// Mitsubishi GX Works2 project: BookEX6_48 Analog   PLC: Q13UDV

// global labels: Global
VAR_GLOBAL
  bVar0 AT M5000 : BOOL;
  abArray0 AT M5010 : ARRAY [0..49] OF BOOL;
  sStr0 AT D5000 : STRING[199];
  sStr1 AT D5100 : STRING[199];
  sStr2 AT D5200 : STRING[199];
  sStr3 AT D5300 : STRING[199];
  sStr4 AT D5400 : STRING[199];
  sStr5 AT D5500 : STRING[199];
  sStr6 AT D5600 : STRING[199];
  sStr7 AT D5700 : STRING[199];
  sStr8 AT D5800 : STRING[199];
  sStr9 AT D5900 : STRING[199];
  iVar0 AT D4500 : INT;
  iVar1 AT D4501 : INT;
  iVar2 AT D4502 : INT;
  iVar3 AT D4503 : INT;
  iVar4 AT D4504 : INT;
  iVar5 AT D4505 : INT;
  iVar6 AT D4506 : INT;
  iVar7 AT D4507 : INT;
  iVar8 AT D4508 : INT;
  iVar9 AT D4509 : INT;
  dVar0 AT D4510 : DINT;
  dVar1 AT D4512 : DINT;
  dVar2 AT D4514 : DINT;
  dVar3 AT D4516 : DINT;
  dVar4 AT D4518 : DINT;
  dVar5 AT D4520 : DINT;
  dVar6 AT D4522 : DINT;
  dVar7 AT D4524 : DINT;
  dVar8 AT D4526 : DINT;
  dVar9 AT D4528 : DINT;
  wVar0 AT D4530 : WORD;
  wVar1 AT D4531 : WORD;
  wVar2 AT D4532 : WORD;
  wVar3 AT D4533 : WORD;
  wVar4 AT D4534 : WORD;
  wVar5 AT D4535 : WORD;
  wVar6 AT D4536 : WORD;
  wVar7 AT D4537 : WORD;
  wVar8 AT D4538 : WORD;
  wVar9 AT D4539 : WORD;
  dwVar0 AT D4540 : DWORD;
  dwVar1 AT D4542 : DWORD;
  dwVar2 AT D4544 : DWORD;
  dwVar3 AT D4546 : DWORD;
  dwVar4 AT D4548 : DWORD;
  dwVar5 AT D4550 : DWORD;
  dwVar6 AT D4552 : DWORD;
  dwVar7 AT D4554 : DWORD;
  dwVar8 AT D4556 : DWORD;
  dwVar9 AT D4558 : DWORD;
  fsVar0 AT D4560 : REAL;
  fsVar1 AT D4562 : REAL;
  fsVar2 AT D4564 : REAL;
  fsVar3 AT D4566 : REAL;
  fsVar4 AT D4568 : REAL;
  fsVar5 AT D4570 : REAL;
  fsVar6 AT D4572 : REAL;
  fsVar7 AT D4574 : REAL;
  fsVar8 AT D4576 : REAL;
  fsVar9 AT D4578 : REAL;
  fdVar0 AT D4580 : LREAL;
  tTime0 AT D4620 : TIME;
  tTime1 AT D4622 : TIME;
  tTime2 AT D4624 : TIME;
  tTime3 AT D4626 : TIME;
  tTime4 AT D4628 : TIME;
  tTime5 AT D4630 : TIME;
  tTime6 AT D4632 : TIME;
  tTime7 AT D4634 : TIME;
  tTime8 AT D4636 : TIME;
  tTime9 AT D4638 : TIME;
  tTime10 AT D4640 : TIME;
  bVar1 AT M5001 : BOOL;
  bVar2 AT M5002 : BOOL;
  bVar3 AT M5003 : BOOL;
  bVar4 AT M5004 : BOOL;
  bVar5 AT M5005 : BOOL;
  bVar6 AT M5006 : BOOL;
  bVar7 AT M5007 : BOOL;
  bVar8 AT M5008 : BOOL;
  bVar9 AT M5009 : BOOL;
  abArray1 AT M5060 : ARRAY [0..49] OF BOOL;
  abArray2 AT M5110 : ARRAY [0..49] OF BOOL;
  abArray3 AT M5160 : ARRAY [0..49] OF BOOL;
  abArray4 AT M5210 : ARRAY [0..49] OF BOOL;
  abArray5 AT M5260 : ARRAY [0..49] OF BOOL;
  abArray6 AT M5310 : ARRAY [0..49] OF BOOL;
  abArray7 AT M5360 : ARRAY [0..49] OF BOOL;
  abArray8 AT M5410 : ARRAY [0..49] OF BOOL;
  abArray9 AT M5460 : ARRAY [0..49] OF BOOL;
  fdVar1 AT D4584 : LREAL;
  fdVar2 AT D4588 : LREAL;
  fdVar3 AT D4592 : LREAL;
  fdVar4 AT D4596 : LREAL;
  fdVar5 AT D4600 : LREAL;
  fdVar6 AT D4604 : LREAL;
  fdVar7 AT D4608 : LREAL;
  fdVar8 AT D4612 : LREAL;
  fdVar9 AT D4616 : LREAL;
  afsPen0 AT D2000 : ARRAY [0..499] OF REAL;
  afsPen1 AT D3000 : ARRAY [0..499] OF REAL;
END_VAR
// user libraries (not included): HMI

FUNCTION_BLOCK adcRead
VAR_INPUT
  i_StartIO : INT;
  i_NoCh : INT;
  b_Reset : BOOL;
END_VAR
VAR_IN_OUT
  b_InitDone : BOOL;
END_VAR
VAR_OUTPUT
  b_Ready : BOOL;
  b_Error : BOOL;
END_VAR
VAR
  Buffer : ARRAY [0..15] OF WORD;
  bRes : BOOL;
  ix : INT;
  SeqInit : INT;
END_VAR
VAR_INPUT
  b_EN : BOOL;
END_VAR
VAR_OUTPUT
  b_ENO : BOOL;
  aw_Setup : ARRAY [0..7] OF WORD;
  ai_Value : ARRAY [0..7] OF INT;
END_VAR
;
b_ENO := b_EN;
IF NOT b_EN THEN
	RETURN;
END_IF;

(* Status *)
Z0 := i_StartIO * 16;
b_Error := X0FZ0;
b_Ready := X00Z0;

(* Reset *)
IF Y0FZ0 AND NOT b_Error THEN Y0FZ0 := FALSE; END_IF;
IF LDP(TRUE, b_Reset) THEN
	SeqInit := 0;
	b_InitDone := FALSE;
	IF b_Error THEN Y0FZ0 := TRUE; END_IF;
END_IF;

CASE SeqInit OF
	0 : 
		IF NOT b_InitDone AND NOT b_Error AND 1 <= i_NoCh AND  i_NoCh <= 8 THEN
			SeqInit := 1;
		END_IF;
	1 : 
		IF b_Ready THEN
			(* Config Setting Read *)
			bRes := FROM(TRUE , i_StartIO , 20 , 2 , Buffer[0]);
			CASE i_NoCh OF
				2 : 
					aw_Setup[0] := Buffer[0] AND 16#000F;
					aw_Setup[1] := Buffer[0] AND 16#00F0;
				4 : 
					aw_Setup[0] := Buffer[0] AND 16#000F;
					aw_Setup[1] := Buffer[0] AND 16#00F0;
					aw_Setup[2] := Buffer[0] AND 16#0F00;
					aw_Setup[3] := Buffer[0] AND 16#F000;
				8 : 
					aw_Setup[0] := Buffer[0] AND 16#000F;
					aw_Setup[1] := Buffer[0] AND 16#00F0;
					aw_Setup[2] := Buffer[0] AND 16#0F00;
					aw_Setup[3] := Buffer[0] AND 16#F000;
					aw_Setup[4] := Buffer[1] AND 16#000F;
					aw_Setup[5] := Buffer[1] AND 16#00F0;
					aw_Setup[6] := Buffer[1] AND 16#0F00;
					aw_Setup[7] := Buffer[1] AND 16#F000;
			END_CASE;
			SeqInit := 2;
		END_IF;
	2 : 
		b_InitDone := TRUE;
		SeqInit := 100;
END_CASE;

IF b_InitDone AND b_Ready AND X0EZ0 THEN
	bRes := FROM(TRUE , i_StartIO , 11 , 8 , Buffer[0]);
	FOR ix := 0 TO i_NoCh-1 BY 1 DO
		IF (Buffer[ix] AND 16#8000) = 16#8000 THEN
			ai_Value[ix] := -WORD_TO_INT(Buffer[ix] AND 16#7FFF);
		ELSE
			ai_Value[ix] := WORD_TO_INT(Buffer[ix] AND 16#7FFF);
		END_IF;
	END_FOR;
END_IF;
END_FUNCTION_BLOCK

FUNCTION_BLOCK adcRead1Ch
VAR_INPUT
  i_Ch : INT;
END_VAR
VAR
  iStatus : INT;
  bRes : BOOL;
END_VAR
VAR_INPUT
  b_EN : BOOL;
END_VAR
VAR_OUTPUT
  b_ENO : BOOL;
END_VAR
VAR_INPUT
  i_StartIO : INT;
END_VAR
VAR_OUTPUT
  b_Error : BOOL;
  i_ErrNo : INT;
  b_OK : BOOL;
END_VAR
VAR
  bReady : BOOL;
END_VAR
VAR_OUTPUT
  i_Value : INT;
END_VAR
VAR
  bStatus : BOOL;
END_VAR
;
b_ENO := b_EN;
IF NOT b_EN THEN
	b_OK := FALSE;
	b_Error := FALSE;
	i_ErrNo := 0;
	RETURN;
END_IF;
IF i_Ch < 1 OR i_Ch > 8 THEN
	b_OK := FALSE;
	b_Error := TRUE;
	i_Value := 0;
	i_ErrNo := 10;
	RETURN;
END_IF;
	
Z0 := i_StartIO * 16;
b_Error := X0FZ0;
bReady := X00Z0;
FROM(TRUE , i_StartIO , 10 , 1 , iStatus);
TEST(TRUE, iStatus, i_Ch-1, bStatus);

IF bReady  AND bStatus THEN 
	FROM(TRUE , i_StartIO , 10+i_Ch, 1 , iStatus);
	i_Value := iStatus;
	b_OK := TRUE;
	i_ErrNo := 0;
END_IF;
END_FUNCTION_BLOCK

FUNCTION_BLOCK adcScaling
VAR_INPUT
  i_Ch : INT;
END_VAR
VAR
  wStatus : INT;
  bRes : BOOL;
END_VAR
VAR_INPUT
  b_EN : BOOL;
END_VAR
VAR_OUTPUT
  b_ENO : BOOL;
END_VAR
VAR_INPUT
  i_StartIO : INT;
END_VAR
VAR_OUTPUT
  b_Error : BOOL;
  i_ErrNo : INT;
  b_OK : BOOL;
END_VAR
VAR
  bReady : BOOL;
END_VAR
VAR_OUTPUT
  i_ScaleValue : INT;
END_VAR
VAR
  bStatus : BOOL;
END_VAR
VAR_INPUT
  i_Upper : INT;
  i_Lower : INT;
  w_ScaleEn : WORD;
END_VAR
VAR_OUTPUT
  w_ScaleComp : WORD;
END_VAR
VAR
  bResolution : BOOL;
  iRangeData : INT;
  dResolution : DINT;
  dwType : DWORD;
  bCalc : BOOL;
  iDigit : INT;
  dDigit : DINT;
  dUpper : DINT;
  dLower : DINT;
  dScale : DINT;
  dOffset : DINT;
  iType : INT;
  dResult : DINT;
END_VAR
;
b_ENO := b_EN;
IF NOT b_EN THEN
	b_OK := FALSE;
	b_Error := FALSE;
	i_ErrNo := 0;
	RETURN;
END_IF;
IF i_Ch < 1 OR i_Ch > 8 THEN
	b_OK := FALSE;
	b_Error := TRUE;
	i_ScaleValue := 0;
	i_ErrNo := 10;
	RETURN;
END_IF;
	
Z0 := i_StartIO * 16;
b_Error := X0FZ0;
bReady := X00Z0;
bResolution := X08Z0;

IF bReady  THEN 
	DFRO(TRUE , i_StartIO , 20 , 1 , dwType);
	DROR(TRUE, (i_Ch-1)*4, dwType);
	iType := DWORD_TO_INT(dwType AND H0F);
	IF bResolution THEN (*고분해능*)
		IF iType = 4 THEN
					dResolution := 32000;
		ELSIF iType = 5 THEN 
					dResolution := 16000;
		ELSE
					dResolution := 12000;
		END_IF;
	ELSE (*일반분해능*)
		IF iType = 4 THEN dResolution := 8000; ELSE dResolution := 4000; END_IF;
	END_IF;				
	FROM(TRUE , i_StartIO , 10 , 1 , wStatus);
	TEST(TRUE, wStatus, i_Ch-1, bStatus);
	IF bStatus AND dResolution <> 0 THEN 	bCalc := TRUE; ELSE bCalc := FALSE; END_IF;
END_IF;
w_ScaleComp := w_ScaleEn;
IF bCalc THEN
	FROM(TRUE , i_StartIO , 11+i_CH-1 , 1 , iDigit);
	dDigit := INT_TO_DINT(iDigit);
	dUpper := INT_TO_DINT(i_Upper);
	dLower := INT_TO_DINT(i_Lower);
	dScale := (dUpper - dLower) * dDigit;
	IF iType = 4 THEN
		dOffset := (dUpper + dLower) / 2;
	ELSE
		dOffset := dLower;
	END_IF;
	dResult := dScale / dResolution;
	dResult := dResult + dOffset;
	IF dResult < -32768 THEN dResult := -32768; END_IF;
	IF dResult > 32767 THEN dResult := 32767; END_IF;
	i_ScaleValue := DINT_TO_INT(dResult);
	b_OK := TRUE;
	i_ErrNo := 0;
	BSET(TRUE, i_CH-1, w_ScaleComp );
ELSE
	BRST(TRUE, i_CH-1, w_ScaleComp);
END_IF;
END_FUNCTION_BLOCK

FUNCTION_BLOCK adcSetIn
VAR_INPUT
  i_Ch : INT;
  b_Enable : BOOL;
END_VAR
VAR
  Buffer : INT;
  bRes : BOOL;
END_VAR
VAR_INPUT
  b_EN : BOOL;
END_VAR
VAR_OUTPUT
  b_ENO : BOOL;
END_VAR
VAR_INPUT
  i_StartIO : INT;
END_VAR
VAR_OUTPUT
  b_Error : BOOL;
  i_ErrNo : INT;
  b_OK : BOOL;
END_VAR
VAR
  bReady : BOOL;
  bAllCh : BOOL;
  ix : INT;
  wStatus : WORD;
END_VAR
;
b_ENO := b_EN;
IF NOT b_EN THEN
	b_OK := FALSE;
	b_Error := FALSE;
	i_ErrNo := 0;
	RETURN;
END_IF;
bAllCh := i_Ch = 15;
IF NOT bAllCh AND (i_Ch < 1 OR i_Ch > 8) THEN
	b_OK := FALSE;
	b_Error := TRUE;
	i_ErrNo := 10;
	RETURN;
END_IF;
	
Z0 := i_StartIO * 16;
ix := i_Ch-1; 
b_Error := X0FZ0;
bReady := X00Z0;

IF bReady  THEN 
	FROM(TRUE , i_StartIO , 0 , 1 , wStatus);
	IF b_Enable THEN
		IF bAllCh THEN
			wStatus := wStatus AND HFF00;
		ELSE
			BRST(TRUE, ix, wStatus);
		END_IF;
	ELSE
		IF bAllCh THEN
			wStatus := wStatus OR H00FF;
		ELSE
			BSET(TRUE, ix, wStatus);
		END_IF;
	END_IF;	
	TO(TRUE , wStatus, i_StartIO ,  0, 1);
	b_OK := TRUE;
	i_ErrNo := 0;
END_IF;
END_FUNCTION_BLOCK

FUNCTION_BLOCK aOFFGAIN
VAR_INPUT
  i_StartIO : INT;
  i_ChNo : INT;
  b_Set : BOOL;
END_VAR
VAR_OUTPUT
  b_X9 : BOOL;
  b_XA : BOOL;
END_VAR
VAR
  Buffer : ARRAY [0..15] OF WORD;
  bRes : BOOL;
  ix : INT;
  SeqPhase : INT;
END_VAR
VAR_INPUT
  i_Value : INT;
  b_Start : BOOL;
END_VAR
VAR_OUTPUT
  b_XB : BOOL;
  b_XC : BOOL;
  b_Y9 : BOOL;
  b_YA : BOOL;
  b_YB : BOOL;
  b_YC : BOOL;
END_VAR
VAR_INPUT
  b_Offset : BOOL;
END_VAR
VAR
  wChNo : WORD;
  iSetVal : INT;
  bX9 : BOOL;
  bXA : BOOL;
  bXB : BOOL;
  bXC : BOOL;
  bY9 : BOOL;
  bYA : BOOL;
  bYB : BOOL;
  bYC : BOOL;
END_VAR
VAR_OUTPUT
  i_Phase : INT;
END_VAR
VAR
  iMode : INT;
END_VAR
;
(* Status *)
Z0 := i_StartIO * 16;
bX9 := X09Z0;
bXA := X0AZ0;
bXB := X0BZ0;
bXC := X0CZ0;
bY9 := Y09Z0;
bYA := Y0AZ0;
bYB := Y0BZ0;
bYC := Y0CZ0;

CASE SeqPhase OF
	0 : (* wait Start *)
		IF LDP(TRUE, b_Start) THEN
			iMode := 1;
			G_OFFGAN(TRUE, H0C, iMode);
			SeqPhase := 1;
		END_IF;
	1 : (* Set or Stop *)
		IF LDP(TRUE, b_Set) THEN
			bY9 := FALSE;
			SeqPhase := 2;
		ELSIF NOT b_Start THEN
			SeqPhase := 8;
		END_IF;
	2 : (* Set Channel No 1~8 *)
		DECO(TRUE, i_ChNo-1, 3, wChNo);
		IF bXA THEN
			IF b_Offset THEN
				Buffer[0] := wChNo;			
				Buffer[1] := 0;			
			ELSE
				Buffer[0] := 0;			
				Buffer[1] := wChNo;			
			END_IF;	
			bRes := TO(TRUE , Buffer[0], i_StartIO , 22 , 2 );
			bYB := TRUE;
			SeqPhase := 3;
		END_IF;
	3 : (* wait ack *)
		IF bXB THEN
			bYB := FALSE;
			SeqPhase := 4;
		END_IF;			
	4 : (* Set Value -3000~3000 *)
		LIMIT(TRUE, -3000, 3000, i_Value, iSetVal);
		Buffer[0] := INT_TO_WORD(iSetVal);			
		bRes := TO(TRUE , Buffer[0], i_StartIO , 24 , 1 );
		bYC := TRUE;	
		SeqPhase := 5;
	5 :  (* wait ack *)
		IF bXC THEN
			bYC := FALSE;
			SeqPhase := 6;
		END_IF;			
	6 : (* wrte *)
		bYA := TRUE;	
		SeqPhase := 7;
	7 :  (* wait ack *)
		IF NOT bXA THEN
			bYA := FALSE;
			SeqPhase := 1;
		END_IF;			
	8 : (* Exit *)
		iMode := 0;
		G_OFFGAN(TRUE, H0C, iMode);
		SeqPhase := 9;
	9 :	
		bY9 := TRUE;
		SeqPhase := 10;
	10 :  (* wait ack *)
		IF NOT bX9 THEN
			SeqPhase := 0;
			bY9 := FALSE;
		END_IF;
END_CASE;
Y09Z0 := bY9;
Y0AZ0 := bYA;
Y0BZ0 := bYB;
Y0CZ0 := bYC;
b_X9 := bX9;
b_XA := bXA;
b_XB := bXB;
b_XC := bXC;
b_Y9 := bY9;
b_YA := bYA;
b_YB := bYB;
b_YC := bYC;
i_Phase := SeqPhase;
END_FUNCTION_BLOCK

FUNCTION_BLOCK dacReset
VAR_INPUT
  b_Reset : BOOL;
END_VAR
VAR
  Buffer : INT;
  bRes : BOOL;
END_VAR
VAR_INPUT
  b_EN : BOOL;
END_VAR
VAR_OUTPUT
  b_ENO : BOOL;
END_VAR
VAR_INPUT
  i_StartIO : INT;
END_VAR
VAR_OUTPUT
  b_Error : BOOL;
  i_ErrNo : INT;
  b_OK : BOOL;
END_VAR
VAR
  bReady : BOOL;
  bIntReset : BOOL;
END_VAR
;
b_ENO := b_EN;
IF NOT b_EN THEN
	b_OK := FALSE;
	b_Error := FALSE;
	i_ErrNo := 0;
	RETURN;
END_IF;

(* Status *)
Z0 := i_StartIO * 16;
b_Error := X0FZ0;
bReady := X00Z0;

IF bReady  THEN 
	IF b_Error THEN
		b_Error := TRUE;
		FROM(TRUE , i_StartIO , 19 , 1 , i_ErrNo);
		IF b_Reset THEN
			Y0FZ0 := TRUE;
			bIntReset := TRUE;
		END_IF;
	END_IF;
	IF NOT b_Reset THEN
		bIntReset := FALSE;
		Y0FZ0 := FALSE;
		b_OK := FALSE;
	END_IF;
	IF bIntReset AND NOT X0FZ0 THEN
		Y0FZ0 := FALSE;
		b_Error := FALSE;
		i_ErrNo := 0;
		b_OK := TRUE;
		bIntReset := FALSE;
	END_IF;
END_IF;
END_FUNCTION_BLOCK

FUNCTION_BLOCK dacSetOut
VAR_INPUT
  i_Ch : INT;
  b_Enable : BOOL;
END_VAR
VAR
  Buffer : INT;
  bRes : BOOL;
END_VAR
VAR_INPUT
  b_EN : BOOL;
END_VAR
VAR_OUTPUT
  b_ENO : BOOL;
END_VAR
VAR_INPUT
  i_StartIO : INT;
END_VAR
VAR_OUTPUT
  b_Error : BOOL;
  i_ErrNo : INT;
  b_OK : BOOL;
END_VAR
VAR
  bReady : BOOL;
  bAllCh : BOOL;
END_VAR
;
b_ENO := b_EN;
IF NOT b_EN THEN
	b_OK := FALSE;
	b_Error := FALSE;
	i_ErrNo := 0;
	RETURN;
END_IF;
bAllCh := i_Ch = 15;
IF NOT bAllCh AND (i_Ch < 1 OR i_Ch > 8) THEN
	b_OK := FALSE;
	b_Error := TRUE;
	i_ErrNo := 10;
	RETURN;
END_IF;
	
Z0 := i_StartIO * 16;
IF bAllCh THEN Z1 := Z0; ELSE Z1 := Z0+i_Ch-1; END_IF;
b_Error := X0FZ0;
bReady := X00Z0;

IF bReady  THEN 
	IF b_Enable THEN
		IF bAllCh THEN
			K2Y1Z1 := HFF;
		ELSE
			Y1Z1 := TRUE;
		END_IF;
	ELSE
		IF bAllCh THEN
			BKRST(TRUE, Y1Z1, 8); 
		ELSE
			Y1Z1 := FALSE;
		END_IF;
	END_IF;	
	b_OK := TRUE;
	i_ErrNo := 0;
END_IF;
END_FUNCTION_BLOCK

FUNCTION_BLOCK dacWrite
VAR_INPUT
  i_NoCh : INT;
  b_Reset : BOOL;
  ai_Value : ARRAY [0..7] OF INT;
END_VAR
VAR_IN_OUT
  b_InitDone : BOOL;
END_VAR
VAR
  Buffer : ARRAY [0..15] OF WORD;
  bRes : BOOL;
  ix : INT;
  SeqInit : INT;
END_VAR
VAR_INPUT
  b_EN : BOOL;
END_VAR
VAR_OUTPUT
  b_ENO : BOOL;
END_VAR
VAR_INPUT
  i_StartIO : INT;
END_VAR
VAR_OUTPUT
  b_Error : BOOL;
  aw_Setup : ARRAY [0..7] OF WORD;
  b_Ready : BOOL;
END_VAR
VAR
  bReset : BOOL;
END_VAR
;
b_ENO := b_EN;
IF NOT b_EN THEN
	RETURN;
END_IF;

Z0 := i_StartIO * 16;
b_Error := X0FZ0;
b_Ready := X00Z0;

IF Y0FZ0 AND NOT b_Error THEN Y0FZ0 := FALSE; END_IF;
IF LDP(TRUE, b_Reset) THEN
	SeqInit := 0;
	b_InitDone := FALSE;
	IF b_Error THEN Y0FZ0 := TRUE; END_IF;
END_IF;

CASE SeqInit OF
	0 : 
		IF NOT b_InitDone AND NOT b_Error AND 1 <= i_NoCh AND i_NoCh <= 8 THEN
			SeqInit := 1;
			Y09Z0 := FALSE;	
		END_IF;
	1 : 
		IF b_Ready AND X09Z0 THEN
			Buffer[0] := 0;			(*변환금지*)
			bRes := TO(TRUE , Buffer[0], i_StartIO , 0 , 1 );
			Y09Z0 := TRUE;		(*설정요구*)
			SeqInit := 2;
		END_IF;
	2 : 
		IF NOT X09Z0 THEN
			Y09Z0 := FALSE;
			SeqInit := 3;
		END_IF;
	3 : 
		IF b_Ready THEN
			bRes := FROM(TRUE , i_StartIO , 20 , 2 , Buffer[0]);
			CASE i_NoCh OF
				2 : 
					Y01Z0 := TRUE;
					Y02Z0 := TRUE;
					aw_Setup[0] := Buffer[0] AND 16#000F;
					aw_Setup[1] := SHR(Buffer[0] AND 16#00F0 , 4);
				4 : 
					Y01Z0 := TRUE;
					Y02Z0 := TRUE;
					Y03Z0 := TRUE;
					Y04Z0 := TRUE;
					aw_Setup[0] := Buffer[0] AND 16#000F;
					aw_Setup[1] := SHR(Buffer[0] AND 16#00F0 , 4);
					aw_Setup[2] := SHR(Buffer[0] AND 16#0F00 , 8);
					aw_Setup[3] := SHR(Buffer[0] AND 16#F000 , 12);
				8 : 
					Y01Z0 := TRUE;
					Y02Z0 := TRUE;
					Y03Z0 := TRUE;
					Y04Z0 := TRUE;
					Y05Z0 := TRUE;
					Y06Z0 := TRUE;
					Y07Z0 := TRUE;
					Y08Z0 := TRUE;
					aw_Setup[0] := Buffer[0] AND 16#000F;
					aw_Setup[1] := SHR(Buffer[0] AND 16#00F0 , 4);
					aw_Setup[2] := SHR(Buffer[0] AND 16#0F00 , 8);
					aw_Setup[3] := SHR(Buffer[0] AND 16#F000 , 12);
					aw_Setup[4] := Buffer[1] AND 16#000F;
					aw_Setup[5] := SHR(Buffer[1] AND 16#00F0 , 4);
					aw_Setup[6] := SHR(Buffer[1] AND 16#0F00 , 8);
					aw_Setup[7] := SHR(Buffer[1] AND 16#F000 , 12);
			END_CASE;
			SeqInit := 4;
		END_IF;
	4 : 
		b_InitDone := TRUE;
		SeqInit := 100;
END_CASE;
IF b_InitDone AND b_Ready THEN
	IF b_Error THEN
		FOR ix := 0 TO i_NoCh-1 BY 1 DO
			Buffer[ix] := 0;
		END_FOR;
		bRes := TO(TRUE , Buffer[0], i_StartIO , 1 , i_NoCh);
	ELSE
		FOR ix := 0 TO i_NoCh-1 BY 1 DO
			Buffer[ix] :=  INT_TO_WORD(ai_Value[ix]);
		END_FOR;
		bRes := TO(TRUE , Buffer[0], i_StartIO , 1 , i_NoCh);
	END_IF;
END_IF;
END_FUNCTION_BLOCK

FUNCTION_BLOCK dacWrite1Ch
VAR_INPUT
  i_Ch : INT;
  i_Value : INT;
END_VAR
VAR
  Buffer : INT;
  bRes : BOOL;
END_VAR
VAR_INPUT
  b_EN : BOOL;
END_VAR
VAR_OUTPUT
  b_ENO : BOOL;
END_VAR
VAR_INPUT
  i_StartIO : INT;
END_VAR
VAR_OUTPUT
  b_Error : BOOL;
  i_ErrNo : INT;
  b_OK : BOOL;
END_VAR
VAR
  bReady : BOOL;
END_VAR
;
b_ENO := b_EN;
IF NOT b_EN THEN
	b_OK := FALSE;
	b_Error := FALSE;
	i_ErrNo := 0;
	RETURN;
END_IF;
IF i_Ch < 1 OR i_Ch > 8 THEN
	b_OK := FALSE;
	b_Error := TRUE;
	i_ErrNo := 10;
	RETURN;
END_IF;
	
Z0 := i_StartIO * 16;
b_Error := X0FZ0;
bReady := X00Z0;

IF bReady  THEN 
	TO(TRUE , i_Value, i_StartIO ,  i_Ch, 1);
	b_OK := TRUE;
	i_ErrNo := 0;
END_IF;
END_FUNCTION_BLOCK

PROGRAM ExLIB
VAR
  dacWrite1Ch_1 : dacWrite1Ch;
  bOK : BOOL;
  bError : BOOL;
  iErrNo : INT;
  dacSetOut_1 : dacSetOut;
  dacWrite_1 : dacWrite;
  daValue : ARRAY [0..7] OF INT;
  waSetup : ARRAY [0..7] OF WORD;
  bInit : BOOL;
  dacReset_1 : dacReset;
  iErrNo2 : INT;
  bError2 : BOOL;
  bOK2 : BOOL;
  adcRead1Ch_1 : adcRead1Ch;
  iCH1 : INT;
  bOK5 : BOOL;
  bError5 : BOOL;
  iErrNo5 : INT;
  adcSetIn_1 : adcSetIn;
  adcScaling_1 : adcScaling;
  bOK6 : BOOL;
  bError6 : BOOL;
  iErrNo6 : INT;
END_VAR
(* structured ladder/FBD written out as ST: instructions are called as NAME(EN, inputs, outputs); _pN, _eN, _tN stand for wires *)
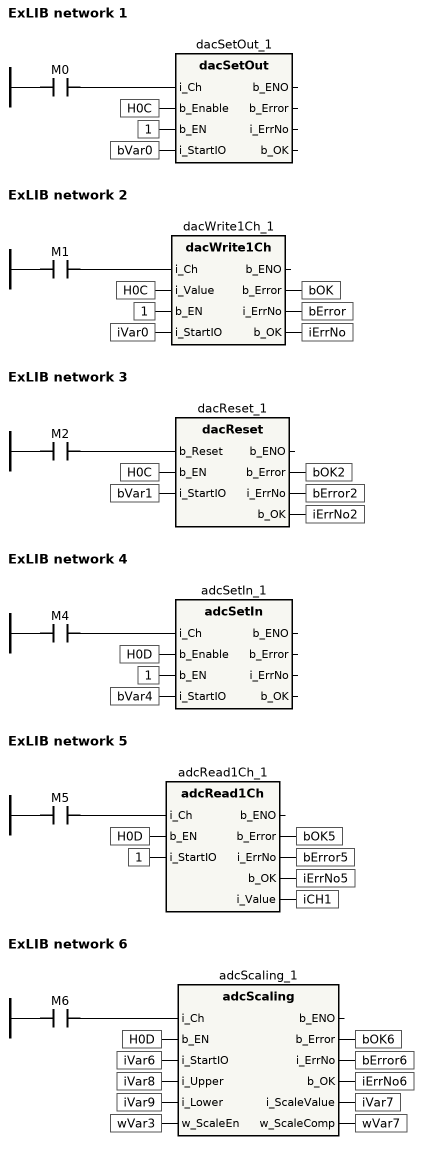
(* network 1 *)
dacSetOut_1(i_Ch := M0, b_Enable := H0C, b_EN := 1, i_StartIO := bVar0);
(* network 2 *)
dacWrite1Ch_1(i_Ch := M1, i_Value := H0C, b_EN := 1, i_StartIO := iVar0, b_Error => bOK, i_ErrNo => bError, b_OK => iErrNo);
(* network 3 *)
dacReset_1(b_Reset := M2, b_EN := H0C, i_StartIO := bVar1, b_Error => bOK2, i_ErrNo => bError2, b_OK => iErrNo2);
(* network 4 *)
adcSetIn_1(i_Ch := M4, b_Enable := H0D, b_EN := 1, i_StartIO := bVar4);
(* network 5 *)
adcRead1Ch_1(i_Ch := M5, b_EN := H0D, i_StartIO := 1, b_Error => bOK5, i_ErrNo => bError5, b_OK => iErrNo5, i_Value => iCH1);
(* network 6 *)
adcScaling_1(i_Ch := M6, b_EN := H0D, i_StartIO := iVar6, i_Upper := iVar8, i_Lower := iVar9, w_ScaleEn := wVar3, b_Error => bOK6, i_ErrNo => bError6, b_OK => iErrNo6, i_ScaleValue => iVar7, w_ScaleComp => wVar7);
END_PROGRAM

PROGRAM ExOFFGAN
VAR
  bFlag : BOOL;
  iMode : INT;
  bSetMode : BOOL;
  bNormalMode : BOOL;
END_VAR
(* structured ladder/FBD written out as ST: instructions are called as NAME(EN, inputs, outputs); _pN, _eN, _tN stand for wires *)
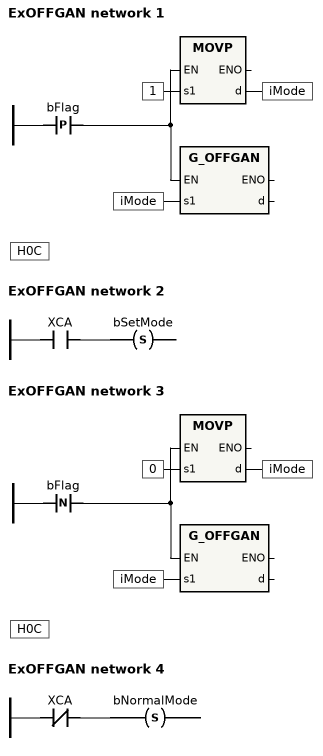
(* network 1 *)
_p1 := LDP(TRUE, bFlag);
MOVP(_p1, 1, iMode);
G_OFFGAN(_p1, iMode, _open);
(* not connected to any output: H0C *)
(* network 2 *)
SET(XCA, bSetMode);
(* network 3 *)
_p1 := LDF(TRUE, bFlag);
MOVP(_p1, 0, iMode);
G_OFFGAN(_p1, iMode, _open);
(* not connected to any output: H0C *)
(* network 4 *)
SET(NOT XCA, bNormalMode);
END_PROGRAM

PROGRAM ExOFFGAN_LD
VAR
  iMode : INT;
  bModeChg : BOOL;
  bChSet : BOOL;
  iChNo : INT;
  bOffset : BOOL;
  bGain : BOOL;
  bAdjust : BOOL;
  bAdjustData : BOOL;
  iAdjustData : INT;
  bAdjustCmd : BOOL;
  bAdjustWrite : BOOL;
  bReturn : BOOL;
END_VAR
(* structured ladder/FBD written out as ST: instructions are called as NAME(EN, inputs, outputs); _pN, _eN, _tN stand for wires *)
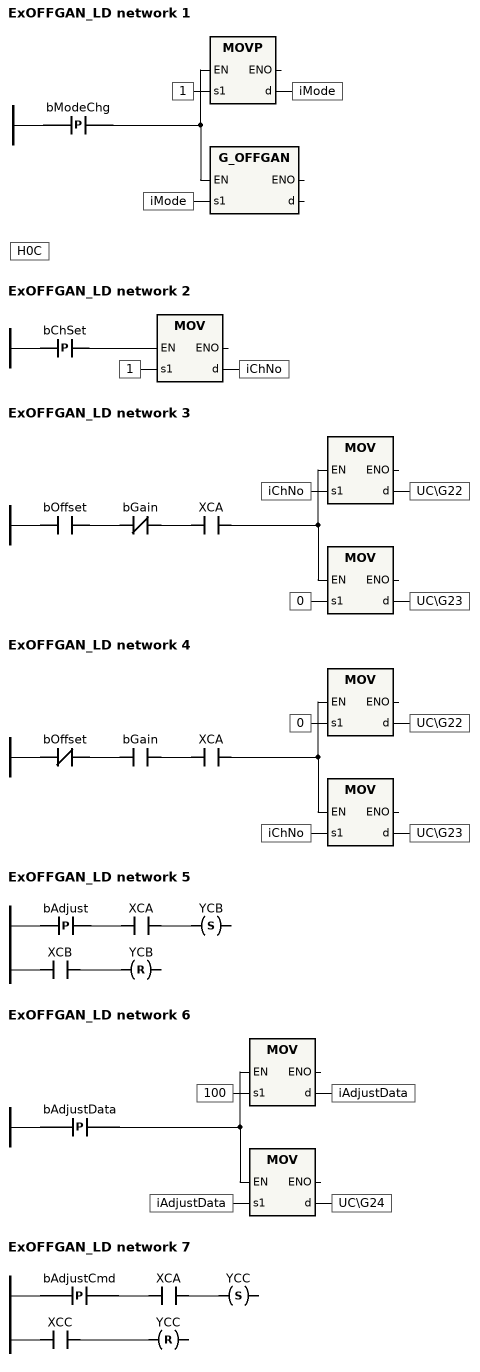
(* network 1 *)
_p1 := LDP(TRUE, bModeChg);
MOVP(_p1, 1, iMode);
G_OFFGAN(_p1, iMode, _open);
(* not connected to any output: H0C *)
(* network 2 *)
MOV(LDP(TRUE, bChSet), 1, iChNo);
(* network 3 *)
_p1 := bOffset AND NOT bGain AND XCA;
MOV(_p1, iChNo, UC\G22);
MOV(_p1, 0, UC\G23);
(* network 4 *)
_p1 := NOT bOffset AND bGain AND XCA;
MOV(_p1, 0, UC\G22);
MOV(_p1, iChNo, UC\G23);
(* network 5 *)
SET(LDP(TRUE, bAdjust) AND XCA, YCB);
RST(XCB, YCB);
(* network 6 *)
_p1 := LDP(TRUE, bAdjustData);
MOV(_p1, 100, iAdjustData);
MOV(_p1, iAdjustData, UC\G24);
(* network 7 *)
SET(LDP(TRUE, bAdjustCmd) AND XCA, YCC);
RST(XCC, YCC);
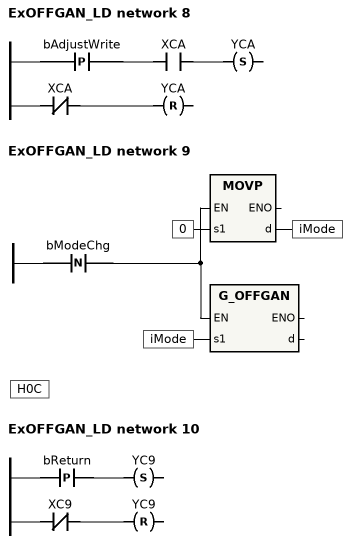
(* network 8 *)
SET(LDP(TRUE, bAdjustWrite) AND XCA, YCA);
RST(NOT XCA, YCA);
(* network 9 *)
_p1 := LDF(TRUE, bModeChg);
MOVP(_p1, 0, iMode);
G_OFFGAN(_p1, iMode, _open);
(* not connected to any output: H0C *)
(* network 10 *)
SET(LDP(TRUE, bReturn), YC9);
RST(NOT XC9, YC9);
END_PROGRAM

PROGRAM ExOFFGAN_ST
VAR
  aOFFGAIN_1 : aOFFGAIN;
END_VAR
(* structured ladder/FBD written out as ST: instructions are called as NAME(EN, inputs, outputs); _pN, _eN, _tN stand for wires *)
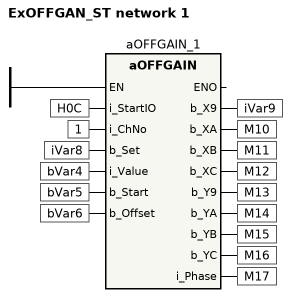
(* network 1 *)
aOFFGAIN_1(EN := TRUE, i_StartIO := H0C, i_ChNo := 1, b_Set := iVar8, i_Value := bVar4, b_Start := bVar5, b_Offset := bVar6, b_X9 => iVar9, b_XA => M10, b_XB => M11, b_XC => M12, b_Y9 => M13, b_YA => M14, b_YB => M15, b_YC => M16, i_Phase => M17);
END_PROGRAM

PROGRAM ExOGLOAD_0C
VAR
  aCtrlData : ARRAY [0..35] OF INT;
  bFlagExe : BOOL;
  abComp : ARRAY [0..1] OF BOOL;
  bError : BOOL;
  bFlag : BOOL;
  bFlag2 : BOOL;
  bFlag2Exe : BOOL;
  abComp2 : ARRAY [0..1] OF BOOL;
  bError2 : BOOL;
END_VAR
(* structured ladder/FBD written out as ST: instructions are called as NAME(EN, inputs, outputs); _pN, _eN, _tN stand for wires *)
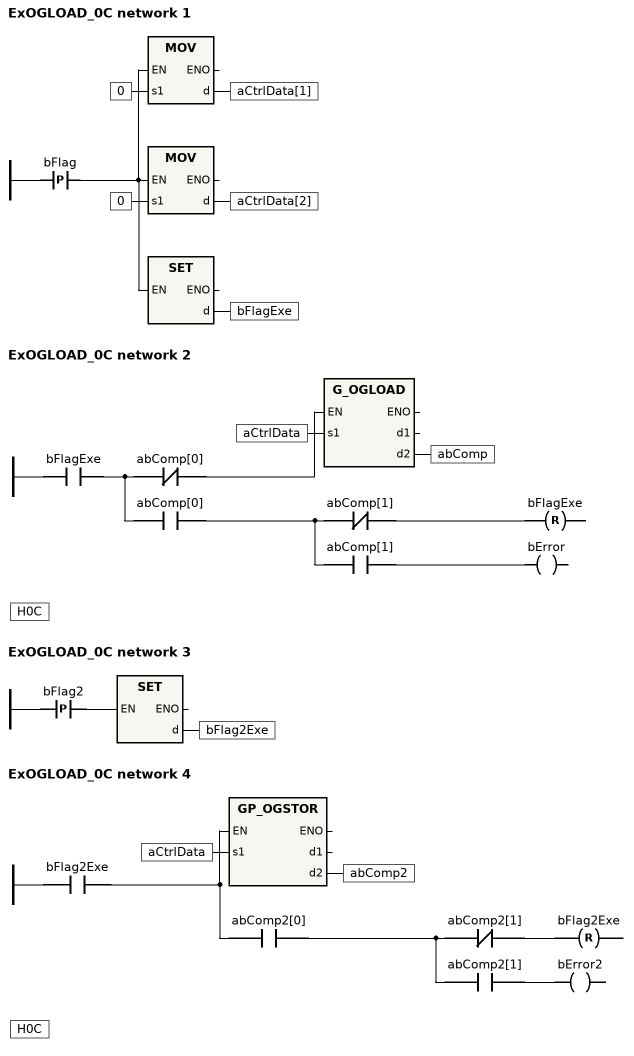
(* network 1 *)
_p1 := LDP(TRUE, bFlag);
MOV(_p1, 0, aCtrlData[1]);
MOV(_p1, 0, aCtrlData[2]);
SET(_p1, bFlagExe);
(* network 2 *)
G_OGLOAD(bFlagExe AND NOT abComp[0], aCtrlData, _open, abComp);
_p1 := bFlagExe AND abComp[0];
RST(_p1 AND NOT abComp[1], bFlagExe);
bError := _p1 AND abComp[1];
(* not connected to any output: H0C *)
(* network 3 *)
SET(LDP(TRUE, bFlag2), bFlag2Exe);
(* network 4 *)
GP_OGSTOR(bFlag2Exe, aCtrlData, _open, abComp2);
_p1 := bFlag2Exe AND abComp2[0];
RST(_p1 AND NOT abComp2[1], bFlag2Exe);
bError2 := _p1 AND abComp2[1];
(* not connected to any output: H0C *)
END_PROGRAM

PROGRAM ExOGLOAD_0D
VAR
  aCtrlData : ARRAY [0..35] OF INT;
  bFlagExe : BOOL;
  abComp : ARRAY [0..1] OF BOOL;
  bError : BOOL;
  bFlag : BOOL;
  bFlag2 : BOOL;
  bFlag2Exe : BOOL;
  abComp2 : ARRAY [0..1] OF BOOL;
  bError2 : BOOL;
END_VAR
(* structured ladder/FBD written out as ST: instructions are called as NAME(EN, inputs, outputs); _pN, _eN, _tN stand for wires *)
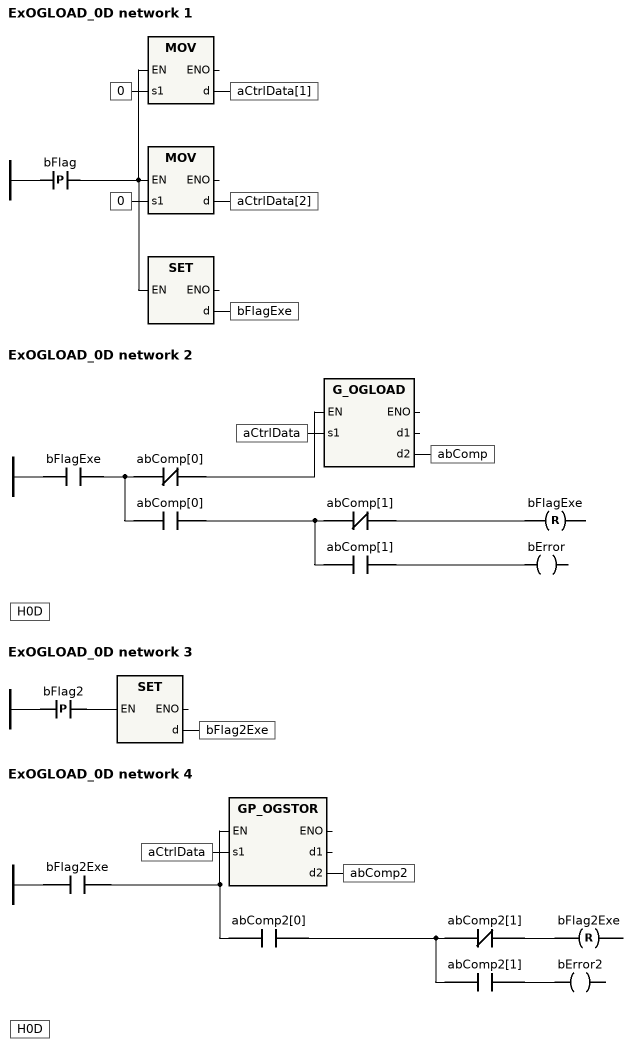
(* network 1 *)
_p1 := LDP(TRUE, bFlag);
MOV(_p1, 0, aCtrlData[1]);
MOV(_p1, 0, aCtrlData[2]);
SET(_p1, bFlagExe);
(* network 2 *)
G_OGLOAD(bFlagExe AND NOT abComp[0], aCtrlData, _open, abComp);
_p1 := bFlagExe AND abComp[0];
RST(_p1 AND NOT abComp[1], bFlagExe);
bError := _p1 AND abComp[1];
(* not connected to any output: H0D *)
(* network 3 *)
SET(LDP(TRUE, bFlag2), bFlag2Exe);
(* network 4 *)
GP_OGSTOR(bFlag2Exe, aCtrlData, _open, abComp2);
_p1 := bFlag2Exe AND abComp2[0];
RST(_p1 AND NOT abComp2[1], bFlag2Exe);
bError2 := _p1 AND abComp2[1];
(* not connected to any output: H0D *)
END_PROGRAM

PROGRAM ExQ64DAN
VAR
  bInit : BOOL;
  bError : BOOL;
  bReady : BOOL;
  bRun : BOOL;
  daValue : ARRAY [0..7] OF INT;
  waSetup : ARRAY [0..7] OF WORD;
  Mov8INT_1 : Mov8INT;
  Mov8WORD_1 : Mov8WORD;
  dacWrite_1 : dacWrite;
  Mov4INT_1 : Mov4INT;
  Mov4WORD_1 : Mov4WORD;
END_VAR
(* structured ladder/FBD written out as ST: instructions are called as NAME(EN, inputs, outputs); _pN, _eN, _tN stand for wires *)
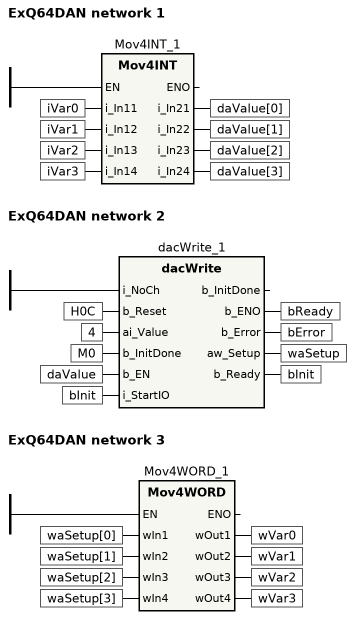
(* network 1 *)
Mov4INT_1(EN := TRUE, i_In11 := iVar0, i_In12 := iVar1, i_In13 := iVar2, i_In14 := iVar3, i_In21 => daValue[0], i_In22 => daValue[1], i_In23 => daValue[2], i_In24 => daValue[3]);
(* network 2 *)
dacWrite_1(i_NoCh := TRUE, b_Reset := H0C, ai_Value := 4, b_InitDone := M0, b_EN := daValue, i_StartIO := bInit, b_ENO => bReady, b_Error => bError, aw_Setup => waSetup, b_Ready => bInit);
(* network 3 *)
Mov4WORD_1(EN := TRUE, wIn1 := waSetup[0], wIn2 := waSetup[1], wIn3 := waSetup[2], wIn4 := waSetup[3], wOut1 => wVar0, wOut2 => wVar1, wOut3 => wVar2, wOut4 => wVar3);
END_PROGRAM

PROGRAM ExQ68ADV
VAR
  bInit : BOOL;
  bError : BOOL;
  bReady : BOOL;
  bRun : BOOL;
  adValue : ARRAY [0..7] OF INT;
  waSetup : ARRAY [0..7] OF WORD;
  dacWrite_1 : dacWrite;
  adcRead_1 : adcRead;
  Mov4INT_1 : Mov4INT;
  Mov4WORD_1 : Mov4WORD;
END_VAR
(* structured ladder/FBD written out as ST: instructions are called as NAME(EN, inputs, outputs); _pN, _eN, _tN stand for wires *)
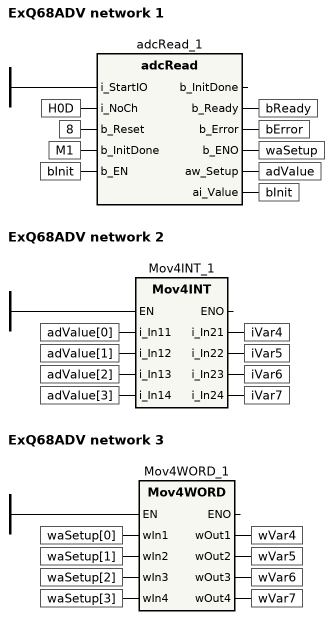
(* network 1 *)
adcRead_1(i_StartIO := TRUE, i_NoCh := H0D, b_Reset := 8, b_InitDone := M1, b_EN := bInit, b_Ready => bReady, b_Error => bError, b_ENO => waSetup, aw_Setup => adValue, ai_Value => bInit);
(* network 2 *)
Mov4INT_1(EN := TRUE, i_In11 := adValue[0], i_In12 := adValue[1], i_In13 := adValue[2], i_In14 := adValue[3], i_In21 => iVar4, i_In22 => iVar5, i_In23 => iVar6, i_In24 => iVar7);
(* network 3 *)
Mov4WORD_1(EN := TRUE, wIn1 := waSetup[0], wIn2 := waSetup[1], wIn3 := waSetup[2], wIn4 := waSetup[3], wOut1 => wVar4, wOut2 => wVar5, wOut3 => wVar6, wOut4 => wVar7);
END_PROGRAM
